(* Ansteuerprogramm der Leitachse. Das Programm hat die Aufgabe, 
   die Leitachse in eine Bewegung konstanter Ge-schwindigkeit zu versetzen, 
   wieder anzuhalten und im Falle eines Fehlers die Achse durch einen Reset 
   wieder in einen funktionstüchtigen Zustand zu versetzen. *)

PROGRAM AufwicklerAnAus
VAR
	//stateMaster				: MoveState_t;		// Programmablauf über Zustandsvariable

	PowerAufwickler				: MC_Power;			// Schaltet Software-Freigabe der Leitachse
	HomeAufwicklerOut: ST_McOutputs;
	PowerAufwicklerOut			: ST_McOutputs;		// 
	
	ResetAufwickler				: MC_Reset;			// Setzt Achsfehler zurück
	ResetAufwicklerOut			: ST_McOutputs;	
	
	MoveAufwickler 				: MC_MoveVelocity;	// Versetzt Leitachse in Bewegung konstanter Geschwindigkeit
	MoveAufwicklerOut			: ST_McOutputs;
	
	HaltAufwickler				: MC_Halt;			// Hält Leitachse an
	GearInAufwicklerOut: ST_McOutputs;
	HaltAufwicklerOut			: ST_McOutputs;
	startAufwicklerTrig: R_TRIG;
	HaltAufwicklerTrig: R_TRIG;
	GearInAufwickler: MC_GearIn;
	GearOutAufwickler: MC_GearOut;
	CamOutAufwicklerOut: ST_McOutputs;
	CamInAufwicklerOut: ST_McOutputs;
	GearOutAufwicklerOut: ST_McOutputs;
	CamInAufwickler: MC_CamIn;
	CamOutAufwickler: MC_CamOut;
	SetCamOnlineChangeMode		: MC_SetCamOnlineChangeMode;				// Legt fest, wann und wie geänderte Kurvenscheibendaten übernommen werden
	SetCamOnlineChangeModeOut	: ST_McOutputs;
	
	CamTableSelect				: MC_CamTableSelect; // Spezifiziert und lädt Kurvenscheibentabelle in die NC
	
	MotionFunction				: ARRAY[1..4] OF MC_MotionFunctionPoint;	// Kurvenscheibe als Motion Function: Eindimensionale Liste (Array) von Stützstellen
	CamTable					: MC_CAM_REF;								// Referenz auf Kurvenscheibe: Beschreibung der Motion Function
	PointID						: MC_MotionFunctionPoint_ID;				// Wird den einzelnen Punkten/Stützstellen der Motion Function zugeordnet
	
	CamInfo						: MC_CamInfo;
	JogAufwicklerOut: ST_McOutputs;
	CamInfoOut					: ST_McOutputs;		
	CamInfoData					: MC_CamInfoData;	
	
	
	JogAufwickler: MC_Jog;
	flag: BOOL;
	AufwicklerHalt: MC_Halt;
	AufwicklerHaltOut: ST_McOutputs;
	HomeAufwickler: MC_Home;
	Kuppelungsmethode: BOOL;
	MARK: INT;
END_VAR

//startAufwicklerTrig(clk := MaschineStart);
//HaltAufwicklerTrig(clk := Abwicklerstopp);

GlobaleVariablen.Aufwickler();
CASE stateAufwickler OF
	
(* ===========================================================================================
   Zustand 1: Programm ist im Ausgangszustand und wartet auf Benutzereingabe. Alle 
   Funktionsbausteine werden initialisiert, etwaige Fehler zurückgesetzt. *)
	MOVESTATE_INIT :

		ResetAufwickler.Execute := FALSE;
		HaltAufwickler.Execute := FALSE;
		PowerAufwickler.Enable := FALSE;
		CamTableSelect.Execute := FALSE;
		CamInAufwickler.Execute := FALSE;
		CamOutAufwickler.Execute := FALSE;
		IF PowerAufwicklerOut.Active THEN
			ResetAufwickler.Execute := TRUE;
			IF ResetAufwickler.Done THEN
				AufwicklerLaeuft := FALSE;
				stateAufwickler := MOVESTATE_INIT;
			END_IF
		END_IF
		//HaltSlave.Execute := FALSE;
		//WriteMotionFunctionPoint.Execute := FALSE;
		//SetCamOnlineChangeMode.ActivationMode := MC_CAMACTIVATION_NEXTCYCLE;
		//SetCamOnlineChangeMode.MasterScalingMode := MC_CAMSCALING_AUTOOFFSET;
		//SetCamOnlineChangeMode.SlaveScalingMode := MC_CAMSCALING_AUTOOFFSET;
		IF AufwicklerStart = TRUE AND MasterLaeuft = FALSE THEN
			stateAufwickler := MOVESTATE_ENABLE;
		ELSIF AufwicklerStart = TRUE AND MasterLaeuft = TRUE THEN
			MasterStopp := TRUE;
		END_IF

(* ===========================================================================================
   Zustand 2: Schlalten der allgemeinen Software-Freigabe, Vorschubfreigabe in positive Richtung
   durch MC_Power. Sobald Funktionsbaustein MC_Power die Betriebsbereitschaft der Achse signalisiert,
   Zustandsübergang in Forward*)
	MOVESTATE_ENABLE :
			PowerAufwickler.Enable := TRUE;
			IF PowerAufwicklerOut.Done THEN
				stateAufwickler := MOVESTATE_HOMING;
			ELSIF PowerAufwickler.Error THEN
				stateAufwickler := MOVESTATE_ERROR;
			END_IF
	MOVESTATE_HOMING:
		IF AufwicklerStart = TRUE AND AufwicklerStopp = FALSE THEN
			HomeAufwickler.Execute := TRUE;

			IF HomeAufwicklerOut.Done THEN
				HomeAufwickler.Execute := FALSE;
				stateAufwickler := MOVESTATE_WRITEMOTIONFUNCTION;
				
			ELSIF HomeAufwicklerOut.CommandAborted OR HomeAufwicklerOut.Error THEN
				stateAufwickler := MOVESTATE_ERROR;
			END_IF
		END_IF	
(* ===========================================================================================
   Zustand 7: Beschreiben der zwei eindimensionalen Arrays mit der Stützstellen der Motion Function. 
   *)	
	MOVESTATE_WRITEMOTIONFUNCTION :
		PointID := 1;												// Dient nur der richtigen Position im Array
			MotionFunction[PointID].PointIndex			:= 1;		// Index der Stützstelle innerhalb der Motion Function
			MotionFunction[PointID].FunctionType 		:= 23;		// Modifizierte Sinuslinie
			MotionFunction[PointID].PointType    		:= 16#0002; // Motion Point Type : Rastpunkt
			MotionFunction[PointID].RelIndexNextPoint 	:= 1;		// Angabe des nächsten Punktes
			MotionFunction[PointID].MasterPos         	:= 0;		// x
			MotionFunction[PointID].SlavePos          	:= 0; 		// psi 
			MotionFunction[PointID].SlaveVelo         	:= 1; 		// psi'
			MotionFunction[PointID].SlaveAcc          	:= 0; 		// psi''
			MotionFunction[PointID].SlaveJerk         	:= 0; 		// psi'''
		
		PointID := 2;
			MotionFunction[PointID].PointIndex			:= 2;		// Polynom 1. Grades -> Gerade in Rast
			MotionFunction[PointID].FunctionType 		:= 23;
			MotionFunction[PointID].PointType    		:= 16#0002;
			MotionFunction[PointID].RelIndexNextPoint 	:= 1;
			MotionFunction[PointID].MasterPos         	:= 120;  	// x
			MotionFunction[PointID].SlavePos          	:= 180;  	// psi 
			MotionFunction[PointID].SlaveVelo         	:= 1; 		// psi'
			MotionFunction[PointID].SlaveAcc          	:= 0; 		// psi''
			MotionFunction[PointID].SlaveJerk         	:= 0; 		// psi'''
			
		PointID := 3;
			MotionFunction[PointID].PointIndex			:= 3;
			MotionFunction[PointID].FunctionType 		:= 23;
			MotionFunction[PointID].PointType    		:= 16#0002;
			MotionFunction[PointID].RelIndexNextPoint 	:= 1;   	// 
			MotionFunction[PointID].MasterPos         	:= 240;		// x
			MotionFunction[PointID].SlavePos          	:= 180;  	// psi 
			MotionFunction[PointID].SlaveVelo         	:= 1;   	// psi'
			MotionFunction[PointID].SlaveAcc          	:= 0; 		// psi''
			MotionFunction[PointID].SlaveJerk         	:= 0; 		// psi'''
			
			
		PointID := 4;
			MotionFunction[PointID].PointIndex			:= 4;
			MotionFunction[PointID].FunctionType 		:= 23;
			MotionFunction[PointID].PointType    		:= 16#0002;
			MotionFunction[PointID].RelIndexNextPoint 	:= 0;   	// 0, da es keinen nächsten Punkt gibt
			MotionFunction[PointID].MasterPos         	:= 360;		// x
			MotionFunction[PointID].SlavePos          	:= 360;  	// psi 
			MotionFunction[PointID].SlaveVelo         	:= 1;   	// psi'
			MotionFunction[PointID].SlaveAcc          	:= 0; 		// psi''
			MotionFunction[PointID].SlaveJerk         	:= 0; 		// psi'''

(*
		PointID := 5;
			MotionFunction[PointID].PointIndex			:= 5;
			MotionFunction[PointID].FunctionType 		:= 1;
			MotionFunction[PointID].PointType    		:= 16#0001;
			MotionFunction[PointID].RelIndexNextPoint 	:= 0;   	// 0, da es keinen nächsten Punkt gibt
			MotionFunction[PointID].MasterPos         	:= x5;		// x
			MotionFunction[PointID].SlavePos          	:= 360;  	// psi 
			MotionFunction[PointID].SlaveVelo         	:= 1;   	// psi'
			MotionFunction[PointID].SlaveAcc          	:= 0; 		// psi''
			MotionFunction[PointID].SlaveJerk         	:= 0; 		// psi'''
			*)
		stateAufwickler := MOVESTATE_CAMTABLESELECT;		
		
		
	(* ===========================================================================================
   Zustand 8: Einlesen, Spezifizieren und in die NC laden der Kurvenscheibendaten. 
   Erste Kurvenscheibe *)	
	MOVESTATE_CAMTABLESELECT :
	
		CamInAufwickler.CamTableID := 1;										 // Festlegung der Kurvenscheiben-ID
		CamTable.TableType := MC_TABLETYPE_MOTIONFUNCTION; 						 // Motion Function und keine Positionstabelle
		CamTable.pArray := ADR(MotionFunction);									 // Adresse des Arrays, der die Stützstellen hält
		CamTable.ArraySize := SIZEOF(MotionFunction);							 // Speichergröße des Arrays
		CamTable.NoOfColumns := 1;												 // Spaltenzahl 
		CamTable.NoOfRows := SIZEOF(MotionFunction) / SIZEOF(MotionFunction[1]); // Zeilenzahl: Gesamtspeicherplatz durch Speicherplatz einer Zeile
		CamTableSelect.Execute := TRUE;
		IF CamTableSelect.Done THEN
			CamTableSelect.Execute := FALSE;
			stateAufwickler := MOVESTATE_CAMIN;
		ELSIF CamTableSelect.Error THEN
			stateAufwickler := MOVESTATE_ERROR;
		END_IF	
		
	MOVESTATE_CAMIN :
		IF AufwicklerStart = TRUE AND AufwicklerStopp = FALSE THEN
			CamInAufwickler.CamTableID := 1;											// Kopplung  mit ID 1
			CamInAufwickler.MasterOffset := 0;										  	// Weder Offset...
			CamInAufwickler.SlaveOffset := 0;
			CamInAufwickler.MasterScaling := 1.0;										// ... noch Skalierung erforderlich
			CamInAufwickler.SlaveScaling := 1.0;
			CamInAufwickler.StartMode := MC_STARTMODE_RELATIVE;						  	// Ursprung des Kurvenscheibenkoordinatensystemes an akt. Achsposition
			CamInAufwickler.Execute := TRUE;
			IF CamInAufwickler.InSync THEN											  	// Kopplung erfolgreich, Kurvenscheibe aktiv
				CamInAufwickler.Execute := FALSE;
				stateAufwickler := MOVESTATE_FORWARD;
			ELSIF CamInAufwickler.CommandAborted OR CamInAufwickler.Error THEN
				stateAufwickler := MOVESTATE_ERROR;
			END_IF
		ELSIF AufwicklerStart = FALSE THEN
			stateAufwickler := MOVESTATE_STOPAUFWICKLER;
		END_IF
		
	MOVESTATE_FORWARD :
		
		IF AufwicklerStart = TRUE AND AufwicklerStopp = FALSE THEN
			AufwicklerLaeuft := TRUE;
			IF AufwicklerJogStart = TRUE THEN
				flag := TRUE;
				stateAufwickler := MOVESTATE_STOPAUFWICKLER;
			END_IF
			IF CamInAufwicklerOut.Done THEN
				AufwicklerLaeuft := TRUE;
			END_IF
		ELSE
			stateAufwickler := MOVESTATE_STOPAUFWICKLER;
		END_IF		

(* ===========================================================================================
   Zustand 4: Anhalten der Leitachse, im Anschluss Rückkehr in den Ausgangszustand. *)		
	MOVESTATE_STOPAUFWICKLER :
		CamOutAufwickler.Execute := TRUE;
		IF CamOutAufwicklerOut.Done THEN
			IF AufwicklerHaltOut.Done THEN	
				AufwicklerHalt.Execute := FALSE;
				IF flag = TRUE AND AufwicklerJogStart = TRUE THEN
					flag := FALSE;
					AufwicklerStopp := FALSE;
					AufwicklerStart := TRUE;
					stateAufwickler := MOVESTATE_JOG;
				ELSE
					AufwicklerStopp := TRUE;
					AufwicklerStart := FALSE;
					AufwicklerLaeuft := FALSE;
					stateAufwickler := MOVESTATE_INIT;
				END_IF
			ELSE
				AufwicklerHalt.Execute := TRUE;
			END_IF
			
			
		ELSIF CamOutAufwickler.Error THEN
			CamOutAufwickler.Execute := FALSE;
			stateAufwickler := MOVESTATE_ERROR;
		END_IF
		
	MOVESTATE_JOG:
		AufwicklerLaeuft := TRUE;
		AufwicklerJoglaeuft := TRUE;
		IF AufwicklerJogStart = FALSE THEN
			AufwicklerJoglaeuft := FALSE;
			stateAufwickler := MOVESTATE_INIT;
		END_IF
	
(* ===========================================================================================
   Zustand 5: Im Falle eines Bausteinfehlers wird überprüft, ob sich die Achse ebenfalls im    
   Fehlerzustand befindet, was einen Achsreset erfordert. Andernfalls werden Bausteinfehler 
   im Zustand Init zurückgesetzt.*)		
	MOVESTATE_ERROR :
		IF Master.Status.Error THEN
			stateAufwickler := MOVESTATE_RESET;	// Reset bei Achsfehler
		ELSE
			stateAufwickler := MOVESTATE_INIT;	// Funktionsbausteinfehler erfordert keinen Reset
		END_IF

(* ===========================================================================================
   Zustand 6:  Durchführung des Achsreset im Fehlerfall  *)		
	MOVESTATE_RESET :
		CamInAufwickler.Execute := FALSE;
		ResetAufwickler.Execute := TRUE;
		IF ResetAufwickler.Done THEN
			AufwicklerLaeuft := FALSE;
			stateAufwickler := MOVESTATE_INIT;
		ELSIF ResetAufwickler.Error THEN
			stateAufwickler := MOVESTATE_INIT; (* Falls Reset nicht gelingt, Benutzereingriff erforderlich *)
		END_IF
		
END_CASE

// Zyklusmäßige Aufrufe
ActPower();		// Aufruf des Power Funktionsbausteines
ActCamming();	// Aufruf des Camming-Funktionsbausteines
ActReset();		// Aufruf des Reset-Funktionsbausteines
ActJog();
ActHalt();
ActHome();

ACTION ActCamming:
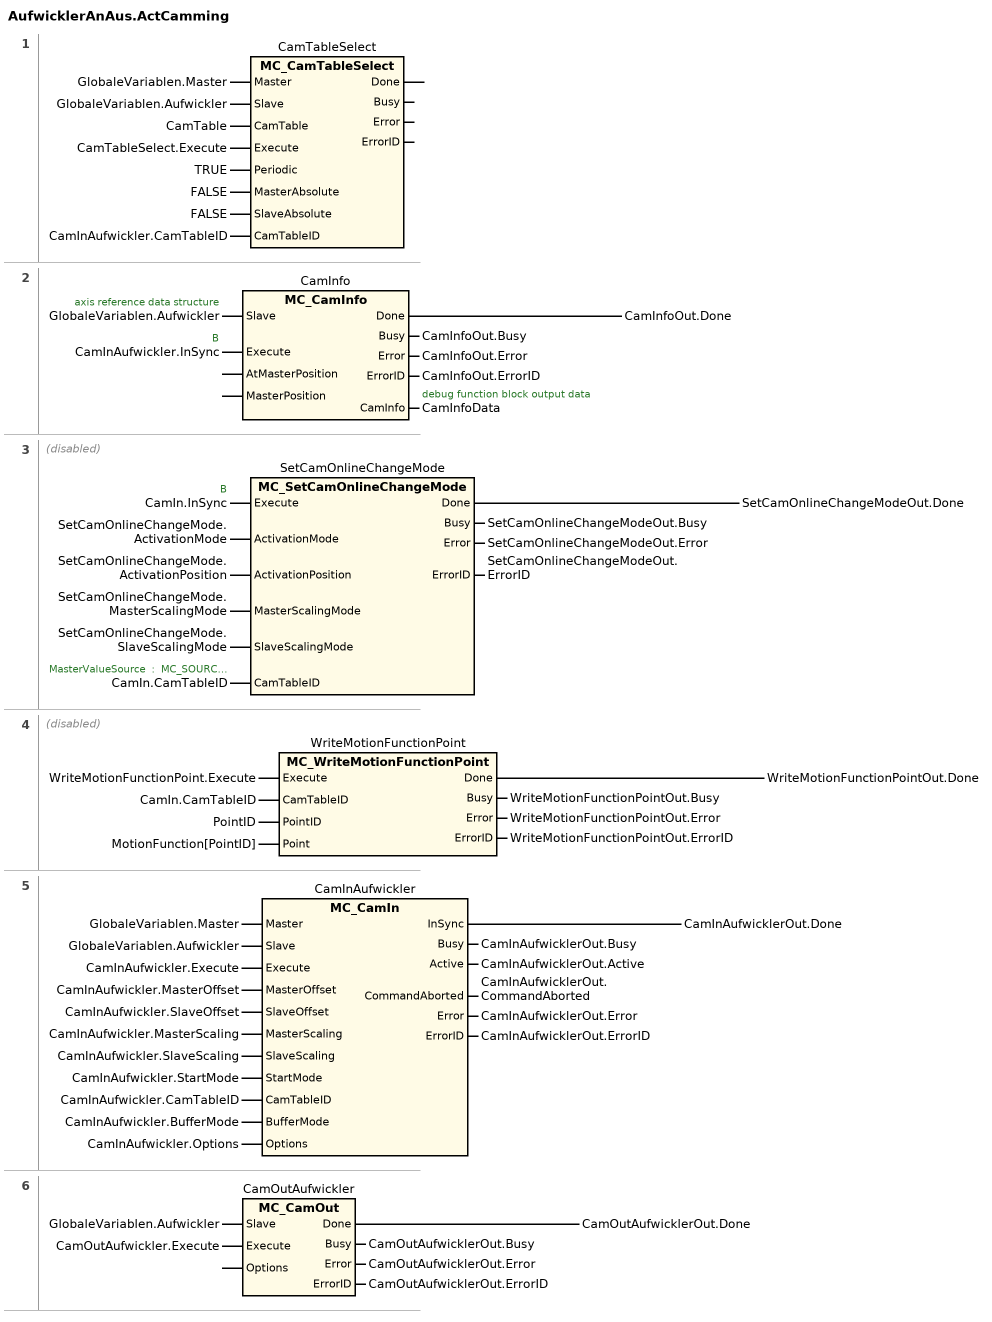
// NETWORK 1
CamTableSelect(
    Master := GlobaleVariablen.Master,
    Slave := GlobaleVariablen.Aufwickler,
    CamTable := CamTable,
    Execute := CamTableSelect.Execute,
    Periodic := TRUE,
    MasterAbsolute := FALSE,
    SlaveAbsolute := FALSE,
    CamTableID := CamInAufwickler.CamTableID); // MC_CamTableSelect

// NETWORK 2
//   GlobaleVariablen.Aufwickler: axis reference data structure
//   CamInAufwickler.InSync: B
//   CamInfoData: debug function block output data
CamInfo(
    Slave := GlobaleVariablen.Aufwickler,
    Execute := CamInAufwickler.InSync,
    Busy => CamInfoOut.Busy,
    Error => CamInfoOut.Error,
    ErrorID => CamInfoOut.ErrorID,
    CamInfo => CamInfoData); // MC_CamInfo
CamInfoOut.Done := CamInfo.Done;

// NETWORK 3 (disabled)
//   CamIn.InSync: B
//   CamIn.CamTableID: MasterValueSource : MC_SOURCE E not available
// SetCamOnlineChangeMode(
//     Execute := CamIn.InSync,
//     ActivationMode := SetCamOnlineChangeMode.ActivationMode,
//     ActivationPosition := SetCamOnlineChangeMode.ActivationPosition,
//     MasterScalingMode := SetCamOnlineChangeMode.MasterScalingMode,
//     SlaveScalingMode := SetCamOnlineChangeMode.SlaveScalingMode,
//     CamTableID := CamIn.CamTableID,
//     Busy => SetCamOnlineChangeModeOut.Busy,
//     Error => SetCamOnlineChangeModeOut.Error,
//     ErrorID => SetCamOnlineChangeModeOut.ErrorID); // MC_SetCamOnlineChangeMode
// SetCamOnlineChangeModeOut.Done := SetCamOnlineChangeMode.Done;

// NETWORK 4 (disabled)
// WriteMotionFunctionPoint(
//     Execute := WriteMotionFunctionPoint.Execute,
//     CamTableID := CamIn.CamTableID,
//     PointID := PointID,
//     Point := MotionFunction[PointID],
//     Busy => WriteMotionFunctionPointOut.Busy,
//     Error => WriteMotionFunctionPointOut.Error,
//     ErrorID => WriteMotionFunctionPointOut.ErrorID); // MC_WriteMotionFunctionPoint
// WriteMotionFunctionPointOut.Done := WriteMotionFunctionPoint.Done;

// NETWORK 5
CamInAufwickler(
    Master := GlobaleVariablen.Master,
    Slave := GlobaleVariablen.Aufwickler,
    Execute := CamInAufwickler.Execute,
    MasterOffset := CamInAufwickler.MasterOffset,
    SlaveOffset := CamInAufwickler.SlaveOffset,
    MasterScaling := CamInAufwickler.MasterScaling,
    SlaveScaling := CamInAufwickler.SlaveScaling,
    StartMode := CamInAufwickler.StartMode,
    CamTableID := CamInAufwickler.CamTableID,
    BufferMode := CamInAufwickler.BufferMode,
    Options := CamInAufwickler.Options,
    Busy => CamInAufwicklerOut.Busy,
    Active => CamInAufwicklerOut.Active,
    CommandAborted => CamInAufwicklerOut.CommandAborted,
    Error => CamInAufwicklerOut.Error,
    ErrorID => CamInAufwicklerOut.ErrorID); // MC_CamIn
CamInAufwicklerOut.Done := CamInAufwickler.InSync;

// NETWORK 6
CamOutAufwickler(
    Slave := GlobaleVariablen.Aufwickler,
    Execute := CamOutAufwickler.Execute,
    Busy => CamOutAufwicklerOut.Busy,
    Error => CamOutAufwicklerOut.Error,
    ErrorID => CamOutAufwicklerOut.ErrorID); // MC_CamOut
CamOutAufwicklerOut.Done := CamOutAufwickler.Done;
END_ACTION

ACTION ActGearInDyn:
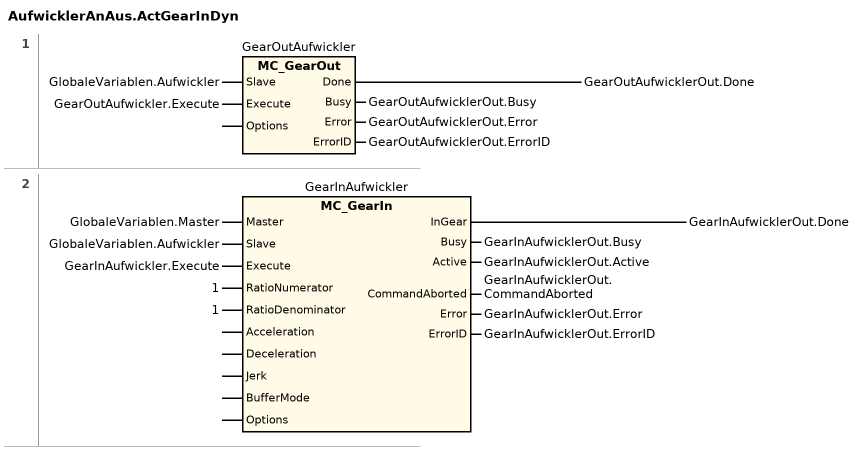
// NETWORK 1
GearOutAufwickler(
    Slave := GlobaleVariablen.Aufwickler,
    Execute := GearOutAufwickler.Execute,
    Busy => GearOutAufwicklerOut.Busy,
    Error => GearOutAufwicklerOut.Error,
    ErrorID => GearOutAufwicklerOut.ErrorID); // MC_GearOut
GearOutAufwicklerOut.Done := GearOutAufwickler.Done;

// NETWORK 2
GearInAufwickler(
    Master := GlobaleVariablen.Master,
    Slave := GlobaleVariablen.Aufwickler,
    Execute := GearInAufwickler.Execute,
    RatioNumerator := 1,
    RatioDenominator := 1,
    Busy => GearInAufwicklerOut.Busy,
    Active => GearInAufwicklerOut.Active,
    CommandAborted => GearInAufwicklerOut.CommandAborted,
    Error => GearInAufwicklerOut.Error,
    ErrorID => GearInAufwicklerOut.ErrorID); // MC_GearIn
GearInAufwicklerOut.Done := GearInAufwickler.InGear;
END_ACTION

ACTION ActHalt:
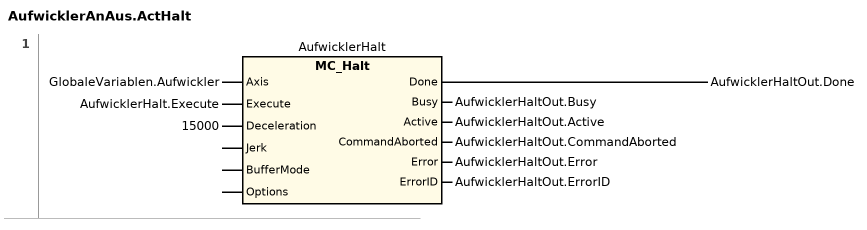
// NETWORK 1
AufwicklerHalt(
    Axis := GlobaleVariablen.Aufwickler,
    Execute := AufwicklerHalt.Execute,
    Deceleration := 15000,
    Busy => AufwicklerHaltOut.Busy,
    Active => AufwicklerHaltOut.Active,
    CommandAborted => AufwicklerHaltOut.CommandAborted,
    Error => AufwicklerHaltOut.Error,
    ErrorID => AufwicklerHaltOut.ErrorID); // MC_Halt
AufwicklerHaltOut.Done := AufwicklerHalt.Done;
END_ACTION

ACTION ActHome:
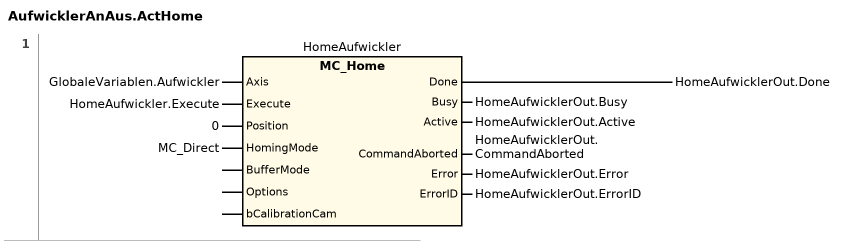
// NETWORK 1
HomeAufwickler(
    Axis := GlobaleVariablen.Aufwickler,
    Execute := HomeAufwickler.Execute,
    Position := 0,
    HomingMode := MC_Direct,
    Busy => HomeAufwicklerOut.Busy,
    Active => HomeAufwicklerOut.Active,
    CommandAborted => HomeAufwicklerOut.CommandAborted,
    Error => HomeAufwicklerOut.Error,
    ErrorID => HomeAufwicklerOut.ErrorID); // MC_Home
HomeAufwicklerOut.Done := HomeAufwickler.Done;
END_ACTION

ACTION ActJog:
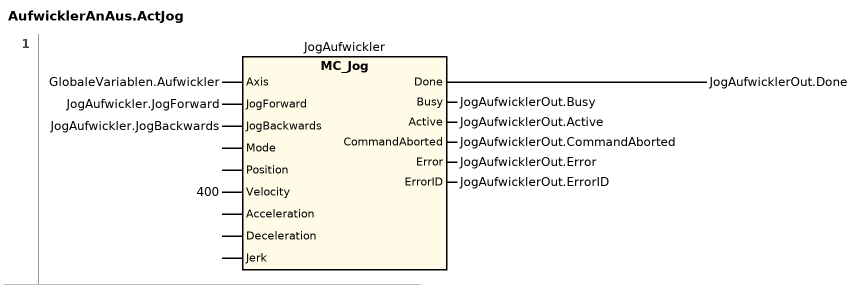
// NETWORK 1
JogAufwickler(
    Axis := GlobaleVariablen.Aufwickler,
    JogForward := JogAufwickler.JogForward,
    JogBackwards := JogAufwickler.JogBackwards,
    Velocity := 400,
    Busy => JogAufwicklerOut.Busy,
    Active => JogAufwicklerOut.Active,
    CommandAborted => JogAufwicklerOut.CommandAborted,
    Error => JogAufwicklerOut.Error,
    ErrorID => JogAufwicklerOut.ErrorID); // MC_Jog
JogAufwicklerOut.Done := JogAufwickler.Done;
END_ACTION

ACTION ActPower:
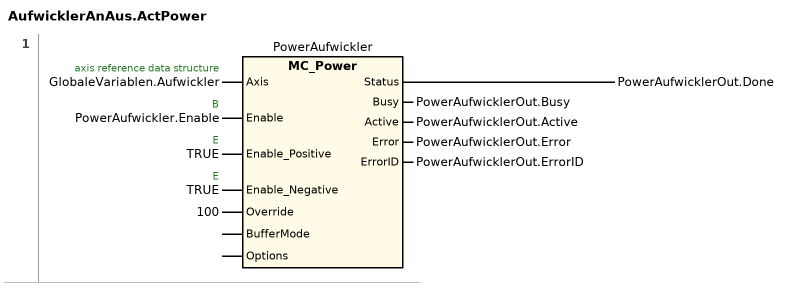
// NETWORK 1
//   GlobaleVariablen.Aufwickler: axis reference data structure
//   PowerAufwickler.Enable: B
//   TRUE: E
PowerAufwickler(
    Axis := GlobaleVariablen.Aufwickler,
    Enable := PowerAufwickler.Enable,
    Enable_Positive := TRUE,
    Enable_Negative := TRUE,
    Override := 100,
    Busy => PowerAufwicklerOut.Busy,
    Active => PowerAufwicklerOut.Active,
    Error => PowerAufwicklerOut.Error,
    ErrorID => PowerAufwicklerOut.ErrorID); // MC_Power
PowerAufwicklerOut.Done := PowerAufwickler.Status;
END_ACTION

ACTION ActReset:
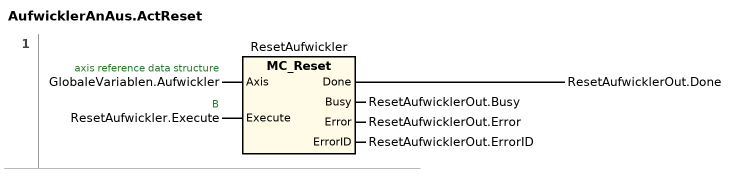
// NETWORK 1
//   GlobaleVariablen.Aufwickler: axis reference data structure
//   ResetAufwickler.Execute: B
ResetAufwickler(
    Axis := GlobaleVariablen.Aufwickler,
    Execute := ResetAufwickler.Execute,
    Busy => ResetAufwicklerOut.Busy,
    Error => ResetAufwicklerOut.Error,
    ErrorID => ResetAufwicklerOut.ErrorID); // MC_Reset
ResetAufwicklerOut.Done := ResetAufwickler.Done;
END_ACTION

END_PROGRAM

(* stored: Version 1.1.0.1, ProductVersion 3.1.4024.11
   POU AufwicklerAnAus: Id {c9892fa9-3be4-4840-ab9e-54b3f2bcc1e3}, SpecialFunc None
   Action ActCamming: Id {0b33aefa-989c-41b7-b80c-3dde86a78f73}
   Action ActGearInDyn: Id {20169739-e56b-4c15-9377-fe7a967efcd8}
   Action ActHalt: Id {65806cdd-0473-456a-b39d-e5bb9aef63e8}
   Action ActHome: Id {0e732bca-c225-4171-818b-134a100084bc}
   Action ActJog: Id {cf02cd48-977b-413d-ad3f-0376dcb6e96e}
   Action ActPower: Id {bf3e3ca8-0cfb-4953-87b4-96443866d170}
   Action ActReset: Id {2cfe771d-4c8a-4c94-9d03-c5b6ee447762} *)
